RoboDK station: Station_2_Bots.rdk

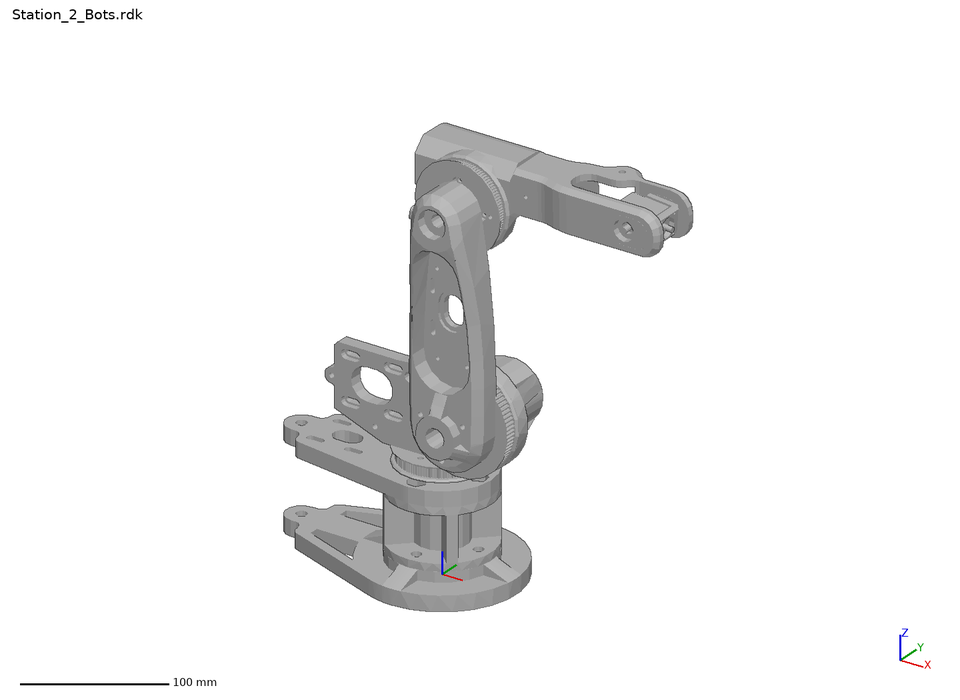
[picture v0: the station drawn from its stored meshes, robots at their saved joint values, targets as dots, program paths as lines]
Station Station_2_Bots (saved by RoboDK 5.9.2). Poses are relative to the parent item; angles as X-Y-Z fixed-axis rotations.
  - frame My Mechanism Base at (145, 1015, 9) mm
    - robot My Mechanism: 6 axes
        modified DH rows (alpha deg, a mm, theta deg, d mm): 0, 0, 0, 135.3; -90, 37.5, -90, 0; 0, 160, 0, 0; -90, 15, 0, 137.3; 90, 0, 0, 0; -90, 0, 180, 0
        joint limits [-200, -200, -200, -200, -200, -200] to [200, 200, 200, 200, 200, 200]; home [0, 0, 0, 0, 0, 0]; saved at [0, 0, 0, 0, 0, 0]
  - frame PartsRefrence at (0, 0, 0) mm
    - object Base at (0, 0, 0) mm, size 187.1 x 120 x 80 mm, geometry from Base.STEP
    - object J1 at (0, 0, 0) mm, size 159.8 x 70 x 95.1 mm, geometry from J1.STEP
    - object J4 at (0, 0, 0) mm, size 122.1 x 56.8 x 36.5 mm, geometry from J4.STEP
    - object J3 at (0, 0, 0) mm, size 78.2 x 55.7 x 80.5 mm, geometry from J3.STEP
    - object J2 at (0, 0, 0) mm, size 79.6 x 44.1 x 219.4 mm, geometry from J2.STEP
    - object J5 at (0, 0, 0) mm, size 31.3 x 37.4 x 24.8 mm, geometry from J5.STEP
    - object J6 at (0, 0, 0) mm, size 41 x 20.5 x 23.2 mm, geometry from J6.STEP
    - frame BaseRef at (145, 15, 9) mm
      - frame ToolRef at (174.8, 0, 310.3) mm, rotated rx 0 ry -90 rz 180 deg
